// SIMATIC S7-200 SMART project (STEP 7-Micro/WIN SMART), CPU CR40

ORGANIZATION_BLOCK MAIN:OB1
TITLE=开始状态M0.0
BEGIN
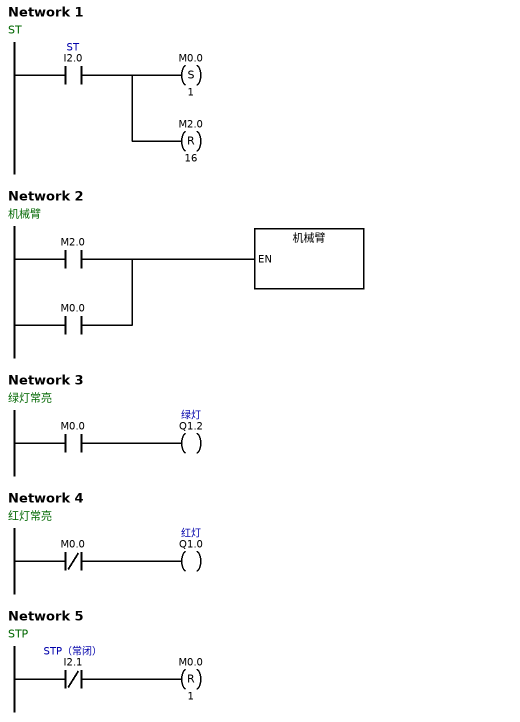
Network 1
// ST
LD     ST:I2.0
S      M0.0, 1
R      M2.0, 16
Network 2
// 机械臂
LD     M2.0
O      M0.0
CALL   机械臂:SBR0
Network 3
// 绿灯常亮
LD     M0.0
=      绿灯:Q1.2
Network 4
// 红灯常亮
LDN    M0.0
=      红灯:Q1.0
Network 5
// STP
LDN    STP（常闭）:I2.1
R      M0.0, 1
END_ORGANIZATION_BLOCK

SUBROUTINE_BLOCK 机械臂:SBR0
TITLE=M2.0：0. 就绪状态，1.工作状态
BEGIN
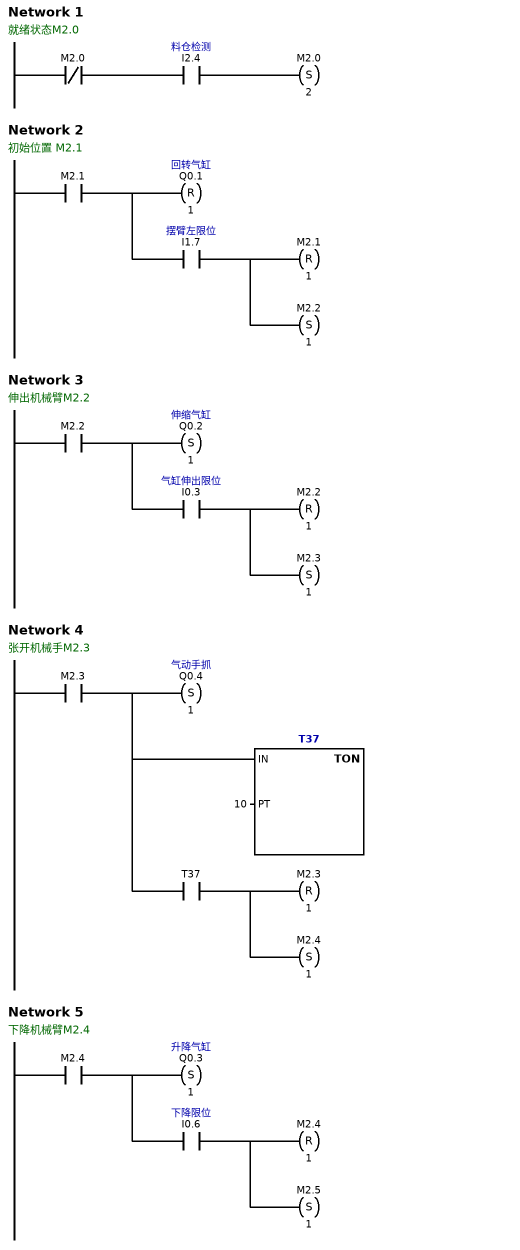
Network 1
// 就绪状态M2.0
LDN    M2.0
A      料仓检测:I2.4
S      M2.0, 2
Network 2
// 初始位置 M2.1
LD     M2.1
R      回转气缸:Q0.1, 1
A      摆臂左限位:I1.7
R      M2.1, 1
S      M2.2, 1
Network 3
// 伸出机械臂M2.2
LD     M2.2
S      伸缩气缸:Q0.2, 1
A      气缸伸出限位:I0.3
R      M2.2, 1
S      M2.3, 1
Network 4
// 张开机械手M2.3
LD     M2.3
S      气动手抓:Q0.4, 1
TON    T37, 10
A      T37
R      M2.3, 1
S      M2.4, 1
Network 5
// 下降机械臂M2.4
LD     M2.4
S      升降气缸:Q0.3, 1
A      下降限位:I0.6
R      M2.4, 1
S      M2.5, 1
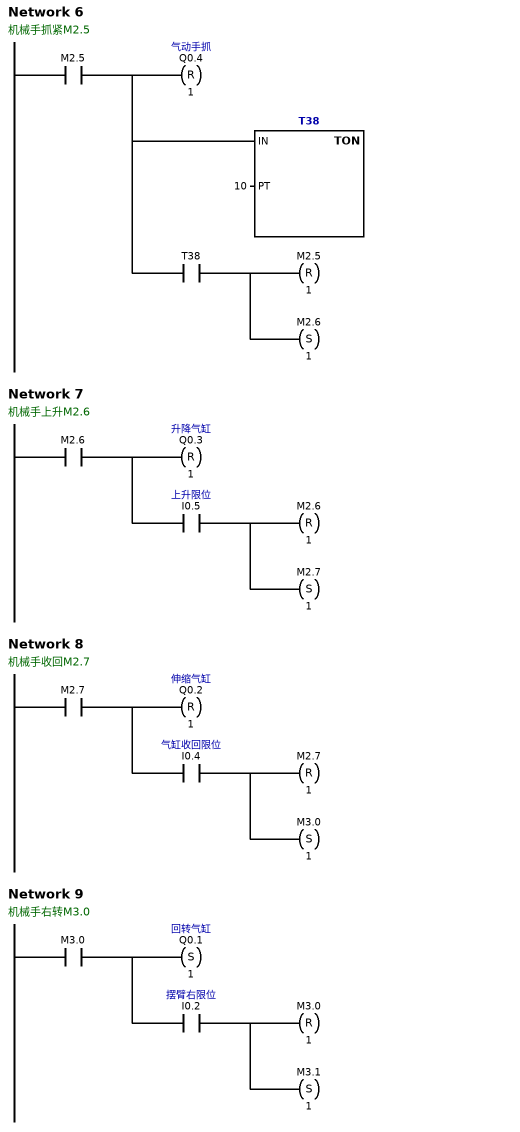
Network 6
// 机械手抓紧M2.5
LD     M2.5
R      气动手抓:Q0.4, 1
TON    T38, 10
A      T38
R      M2.5, 1
S      M2.6, 1
Network 7
// 机械手上升M2.6
LD     M2.6
R      升降气缸:Q0.3, 1
A      上升限位:I0.5
R      M2.6, 1
S      M2.7, 1
Network 8
// 机械手收回M2.7
LD     M2.7
R      伸缩气缸:Q0.2, 1
A      气缸收回限位:I0.4
R      M2.7, 1
S      M3.0, 1
Network 9
// 机械手右转M3.0
LD     M3.0
S      回转气缸:Q0.1, 1
A      摆臂右限位:I0.2
R      M3.0, 1
S      M3.1, 1
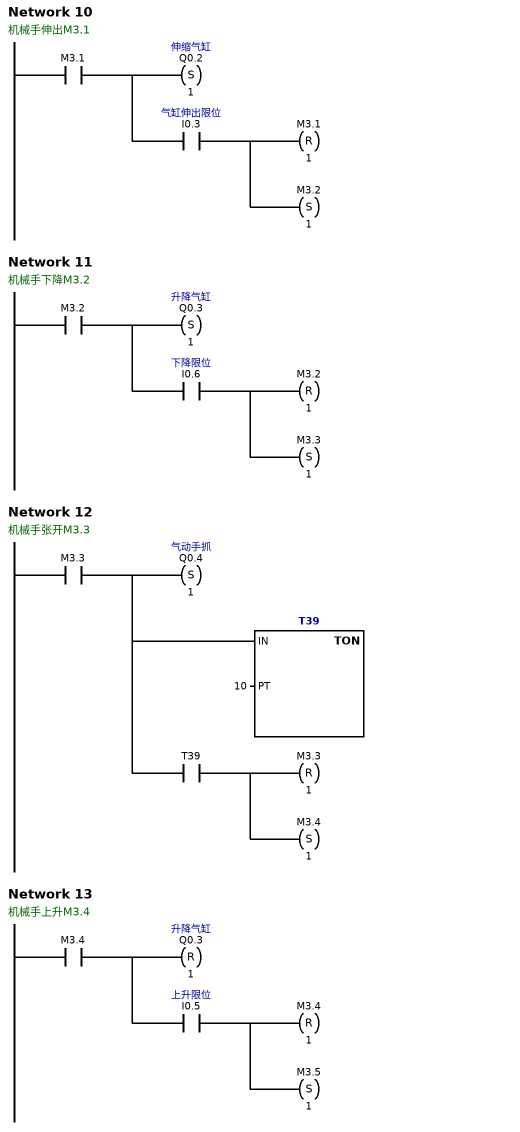
Network 10
// 机械手伸出M3.1
LD     M3.1
S      伸缩气缸:Q0.2, 1
A      气缸伸出限位:I0.3
R      M3.1, 1
S      M3.2, 1
Network 11
// 机械手下降M3.2
LD     M3.2
S      升降气缸:Q0.3, 1
A      下降限位:I0.6
R      M3.2, 1
S      M3.3, 1
Network 12
// 机械手张开M3.3
LD     M3.3
S      气动手抓:Q0.4, 1
TON    T39, 10
A      T39
R      M3.3, 1
S      M3.4, 1
Network 13
// 机械手上升M3.4
LD     M3.4
R      升降气缸:Q0.3, 1
A      上升限位:I0.5
R      M3.4, 1
S      M3.5, 1
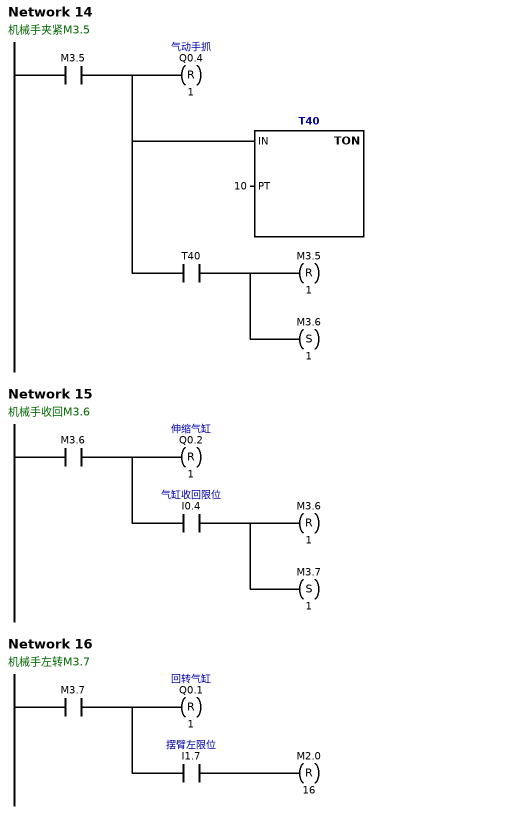
Network 14
// 机械手夹紧M3.5
LD     M3.5
R      气动手抓:Q0.4, 1
TON    T40, 10
A      T40
R      M3.5, 1
S      M3.6, 1
Network 15
// 机械手收回M3.6
LD     M3.6
R      伸缩气缸:Q0.2, 1
A      气缸收回限位:I0.4
R      M3.6, 1
S      M3.7, 1
Network 16
// 机械手左转M3.7
LD     M3.7
R      回转气缸:Q0.1, 1
A      摆臂左限位:I1.7
R      M2.0, 16
END_SUBROUTINE_BLOCK
